// TIA Portal V18 export
DATA_BLOCK "_DEFECT_DB"   // DB44
{ S7_Optimized_Access := 'TRUE' }
VERSION : 0.1
// stored: AutoNumber true, DBAccessibleFromOPCUA true, IsOnlyStoredInLoadMemory false, IsRetainMemResEnabled false, IsWriteProtectedInAS false, MemoryReserve 100
   VAR
      DB : "typeDefectsDB";
   END_VAR
BEGIN
END_DATA_BLOCK
